FUNCTION VisuDlg_CheckedAppend : BOOL
VAR_IN_OUT
	stOutputValue : STRING;
	stVariableValue : STRING;
	bInit : BOOL;
END_VAR
VAR_INPUT
	bPassword : BOOL;
	cToAppend : STRING(1);
END_VAR

DialogCheckInit(stVariableValue, stOutputValue, bInit);

stVariableValue := CONCAT(stVariableValue, cToAppend);
IF bPassword THEN
	stOutputValue := CONCAT(stOutputValue, Dialog_Constants.PASSWORD_CHAR);
ELSE
	stOutputValue := stVariableValue;
END_IF

END_FUNCTION

(* stored: Version 1.1.0.1, ProductVersion 3.1.4024.2
   POU VisuDlg_CheckedAppend: Id {f3c4d79c-83cd-49c5-9525-921dde99184a}, SpecialFunc None *)
